PROGRAM State
VAR
	MemoryCoil: BOOL;
	BreakCondition: BOOL;
	Trigger: BOOL;
	
	//esimerkki ylikuumenemissuojasta
	OverTempFault: BOOL;
	TempOK: BOOL;
	FaultReset: BOOL;
	
END_VAR

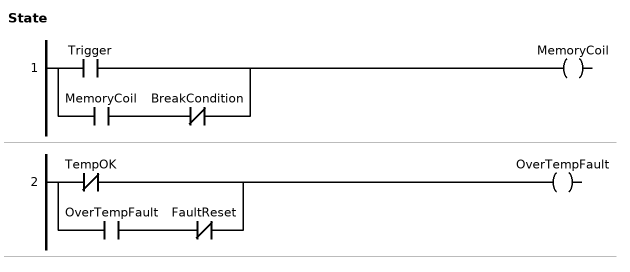
// NETWORK 1
MemoryCoil := Trigger OR MemoryCoil AND NOT BreakCondition;

// NETWORK 2
OverTempFault := NOT TempOK OR OverTempFault AND NOT FaultReset;

END_PROGRAM

(* stored: Version 1.1.0.1, ProductVersion 3.1.4024.10
   POU State: Id {f308e131-9b00-4f4b-b877-5837dd73d1f8}, SpecialFunc None *)
